ABB RobotStudio station: ABB-2600-12-1.85_20211019-085739.rsstn

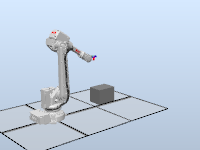
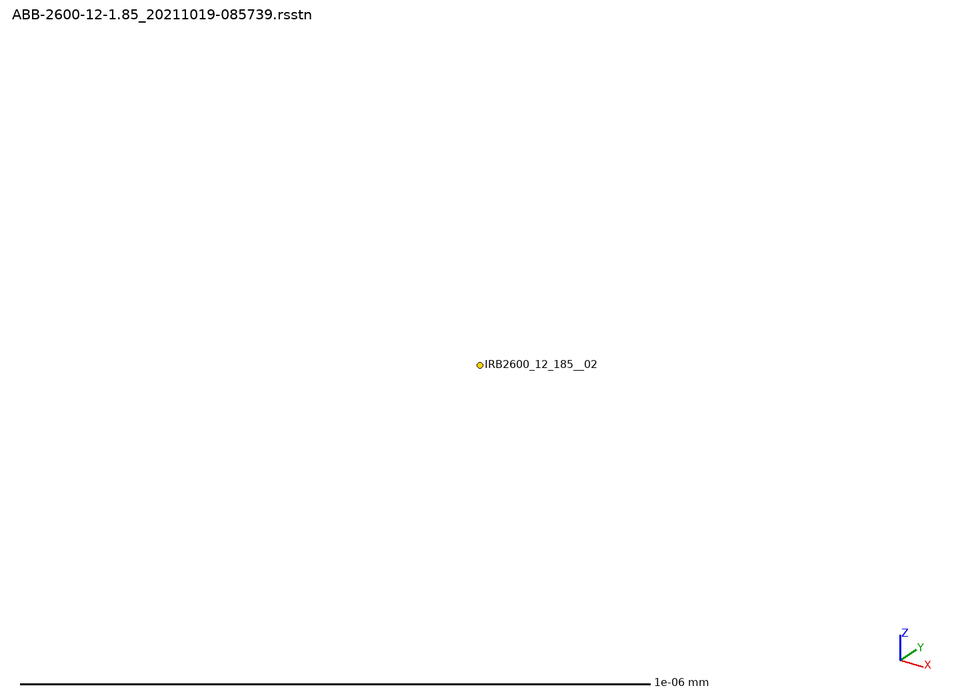
[picture v1: parts stored in the station drawn from their meshes, with robot base, taught points and paths (robot models come from the ABB library and are not in the file)]
Station ABB-2600-12-1.85 (saved by RobotStudio 21.2.9526.0)
Controller IRB2600_12_185
  mechanical unit ROB_1: IRB2600_12_185__02, 6 joints, base frame (0, 0, 0) mm
Layout (positions relative to the parent item):
  - IRB2600_12_185__02 [mechanism, from Robots\IRB2600_12_185_G_02.rslib] at (0, 0, 0) mm; joint values [0.0598, -0.0437, 0.6301, -3.0338, 0.5891, 3.0519] (rad or m)
  - Tool [mechanism] at (920, 50, 1000) mm, rotated rx 0 ry 90 rz 0 deg
      TCP Tool at (0, 0, 80) mm
      links: Tool
  - Part_1 [part], size 400 x 300 x 308 mm
  - Frame_1 [frame] at (0, 0, 80) mm
Attachment: Tool is attached to IRB2600_12_185__02 / Link6
Targets, tools, work objects and paths stored in the station, written as RAPID:
! task T_ROB1
MODULE CalibData
  PERS tooldata Tool:=[TRUE,[[0,0,80],[1,0,0,0]],[1,[0,0,100],[1,0,0,0],0,0,0]];
ENDMODULE

! task T_ROB1
MODULE Module1
  CONST robtarget Target_10:=[[1000,50,1000],[0.707106781,0,0.707106781,0],[0,0,0,0],[9E+09,9E+09,9E+09,9E+09,9E+09,9E+09]];
ENDMODULE

